FUNCTION fc_Floor2 : DINT
VAR_INPUT
	X : REAL;
END_VAR
VAR
END_VAR

fc_Floor2 := REAL_TO_DINT(X);
IF DINT_TO_REAL(fc_Floor2) > X THEN
	fc_Floor2 := fc_Floor2 - 1;
END_IF;

END_FUNCTION

(* stored: Version 1.1.0.1, ProductVersion 3.1.4024.11
   POU fc_Floor2: Id {318c046d-7fdc-46e5-8817-8747fa4d9099}, SpecialFunc None *)
